FUNCTION_BLOCK FB_pushBtnNO
VAR
	bBtn AT %I* : BOOL;
END_VAR

PROPERTY isPressed : BOOL
GET
IF bBtn THEN 
	isPressed := TRUE;
ELSE 
	isPressed := FALSE;
END_IF
END_GET
END_PROPERTY

END_FUNCTION_BLOCK

(* stored: Version 1.1.0.1, ProductVersion 3.1.4024.13
   POU FB_pushBtnNO: Id {de989b08-743c-4971-9daa-f8cb71f34a05}, SpecialFunc None
   Property isPressed: Id {cad453dd-2aec-4160-b392-919d864cba81}
   Get Get: Id {ea29fd4f-6daa-45c9-b910-7c09106f879b} *)
